VAR_GLOBAL
	
END_VAR

(* stored: Version 1.1.0.1, ProductVersion 3.1.4022.9
   GVL Global_Variables: Id {50f738d8-8e33-415b-bcc2-793616d4f251} *)
